(* PLC project Rasi_feeds_batching.project, Automation Builder 2.7 - Basic Automation Builder 2.7 *)
(* stored: creationDateTime 2026-08-29T13:26:29 *)

CONFIGURATION Application
  RESOURCE Application ON PLC
    TASK Task(INTERVAL := T#10ms, PRIORITY := 14);
    PROGRAM batching14 WITH Task : batching14;
  END_RESOURCE
END_CONFIGURATION
